FUNCTION_BLOCK AxisReferencing
VAR_INPUT
	referencingSpeed: INT;
	ReferenceSwitch:BOOL;
END_VAR
VAR_OUTPUT
	AxisPlus:BOOL;
	AxisMinus:BOOL;
	Control:INT;
	SpeedPWM:INT;
	SetCounterValue: UINT;
	SetCounter:BOOL;
	ReferenceOkay:BOOL;
END_VAR
VAR
END_VAR

IF ReferenceSwitch THEN
	AxisMinus := FALSE;
	AxisPlus := FALSE;
	Control := 0;
	SpeedPWM := 0;
	SetCounter := TRUE;
	ReferenceOkay:= TRUE;
ELSE
	AxisMinus := TRUE;
	AxisPlus := FALSE;
	Control := 32;
	SetCounterValue := 0;
	SpeedPWM := referencingSpeed;
	SetCounter := FALSE;
END_IF

END_FUNCTION_BLOCK

(* stored: Version 1.1.0.1, ProductVersion 3.1.4024.12
   POU AxisReferencing: Id {d3500eca-3f04-4172-914d-e4ec9b439d98}, SpecialFunc None *)
